{attribute addProperty BoxType "KL9900-0058"}
{attribute addProperty Id "Channel_1Channel_38696CC400"}
{attribute addProperty CRC "402178980"}
{attribute addProperty SizeInBites "0"}
{attribute addProperty SizeInBytes "0"}
TYPE KL_17F8C3A4 :
STRUCT
	{attribute addProperty Name "Channel_1"}
	Channel_1 : Channel_38696CC4;
END_STRUCT
END_TYPE

(* stored: Version 1.2.0.0, ProductVersion 3.1.4024.9
   DUT KL_17F8C3A4: Id {343805f4-084d-4a49-a689-e53d0b3757da} *)
